Staubli VAL3: network.dtx

bool convnum = true
bool hasmsg
bool isx
bool isy = true
mdesc mNomSpeed
mdesc speed = {accel=9, vel=30, decel=9}
num cont
num divmsg = 5
num endmsg = 11
num gstart
num msg[32]
  [1] = 88
  [2] = 50
  [3] = 53
  [4] = 49
  [5] = 89
  [6] = 45
  [7] = 49
  [8] = 54
  [9] = 55
  [10] = 69
  [11] = 69
  [12] = 69
  [13] = 57
  [14] = 69
num xxx = 251
num yyy = -167
pointRs a = {x=407.52, y=-8.68, z=5.9, rx=-180, ry=-1.455991e-32, rz=-0.24, fatherId=world[0]}
pointRs home = {x=407.53, y=-8.71, z=140.1, rx=-180, ry=-1.412482e-32, rz=-0.23, fatherId=world[0]}
pointRs photo = {x=400, y=375, z=180, rx=-180, fatherId=world[0]}
sio input = {link=Socket\staubli}
string axxx = "251"
string ayyy = "-167"
string endchr = "E"
string message[32]
  [0] = "251-167"
  [1] = "M"
  [2] = "S"
  [3] = "G"
string split = "/"
tool garra = {x=20.5, y=13.05, z=13.77, fatherId=flange[0], ioLink=valve1}
